Omron CX-Programmer project NewProject (CX-Programmer 9.61)

# PLC NewPLC2: CJ2H CPU64

## Global symbols (name address type ; comment)
0.00 BOOL  ; PB ON
0.01 BOOL  ; PB OFF
0.02 BOOL  ; PB COUNT
0.03 BOOL  ; PB COUNT
10.00 BOOL  ; RELAY
10.01 BOOL  ; LAMPU COUNTER

## Program NewProgram1 (cyclic task 0)

### Section Section1

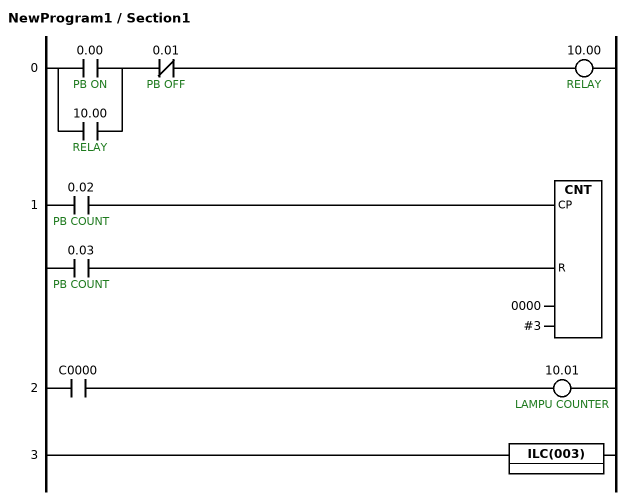
; rung 0
LD 0.00  ; PB ON
OR 10.00  ; RELAY
ANDNOT 0.01  ; PB OFF
OUT 10.00  ; RELAY
; rung 1
LD 0.02  ; PB COUNT
LD 0.03  ; PB COUNT
CNT 0000 #3
; rung 2
LD C0000
OUT 10.01  ; LAMPU COUNTER
; rung 3
ILC(003)

### Section END
; rung 0
END(001)